(* Node for linked list*)
{attribute 'enable_dynamic_creation'}
TYPE ST_NODE:
STRUCT
	Data 	: ST_GENERIC; // Stored data.
	pNext 	: POINTER TO ST_NODE := Tc3_Module.GVL.NULL; 	// Pointer to next node.
END_STRUCT
END_TYPE

(* stored: Version 1.1.0.1, ProductVersion 3.1.4024.4
   DUT ST_NODE: Id {ae72523c-b4d2-4bc3-a909-213c887bca25} *)
